ABB RobotStudio station: Demo Solar Simulation.rspag

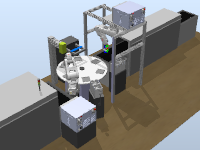
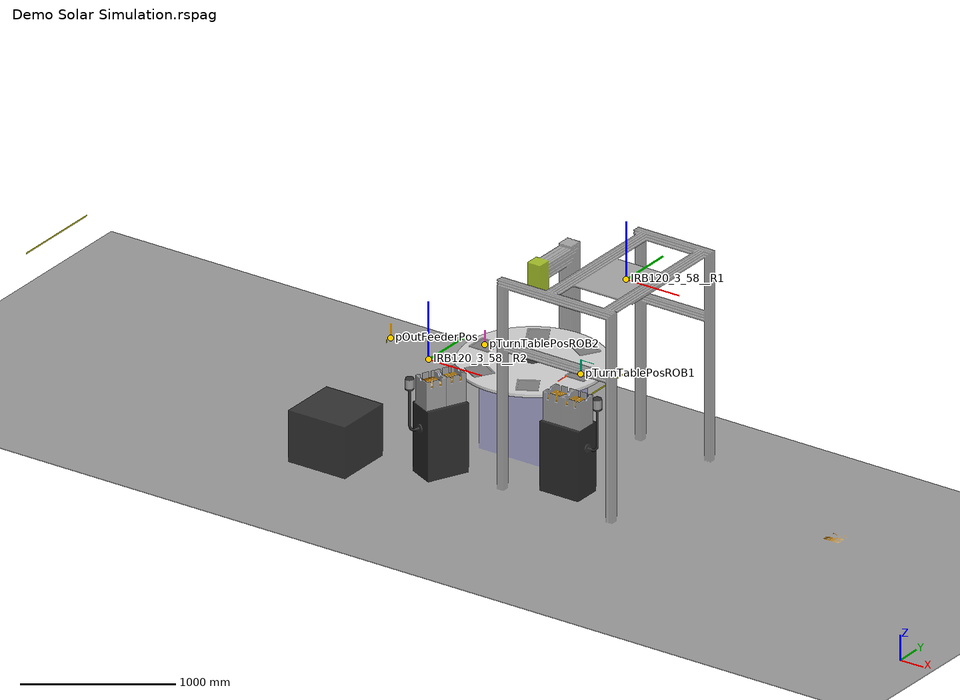
[picture v1: parts stored in the station drawn from their meshes, with robot base, taught points and paths (robot models come from the ABB library and are not in the file)]
--- station ---
Station Demo Solar Simulation (saved by RobotStudio 21.4.9694.0)
Controller IRB120_ROB1, task T_ROB1: task frame (RAPID world) sits at (800, -100, 1439.5) mm, rotated rx 180 ry 0 rz 90 deg in the station
Controller IRB120_ROB2, task T_ROB1: task frame (RAPID world) sits at (-554.4, -372.68, 600) mm, rotated rx 0 ry 0 rz 45 deg in the station
Controller IRB120_ROB2
  mechanical unit ROB_1: IRB120_3_58__R2, 6 joints, base frame (0, 0, 0) mm
Controller IRB120_ROB1
  mechanical unit ROB_1: IRB120_3_58__R1, 6 joints, base frame (0, 0, 0) mm
Layout (positions relative to the parent item):
  - Robotfoot_600 [part, from Libraries\Robotfoot_600.rslib] at (-554.37, -514.08, 0) mm, rotated rx 0 ry 0 rz 45 deg
  - VisionCamStand1 [part] at (-238.48, 626.57, 0) mm, size 100 x 350 x 1120 mm
  - SC_TurnTable [smart component] at (-5618.3, -2219.9, 0) mm
      signals: DI diROB1detached, DI diRotateOK_ROB2, DI diRotateOK_ROB1, DO doTurnTableInPos, DO doCellInPickPosROB2, DO doTurnTableReadyToRotate
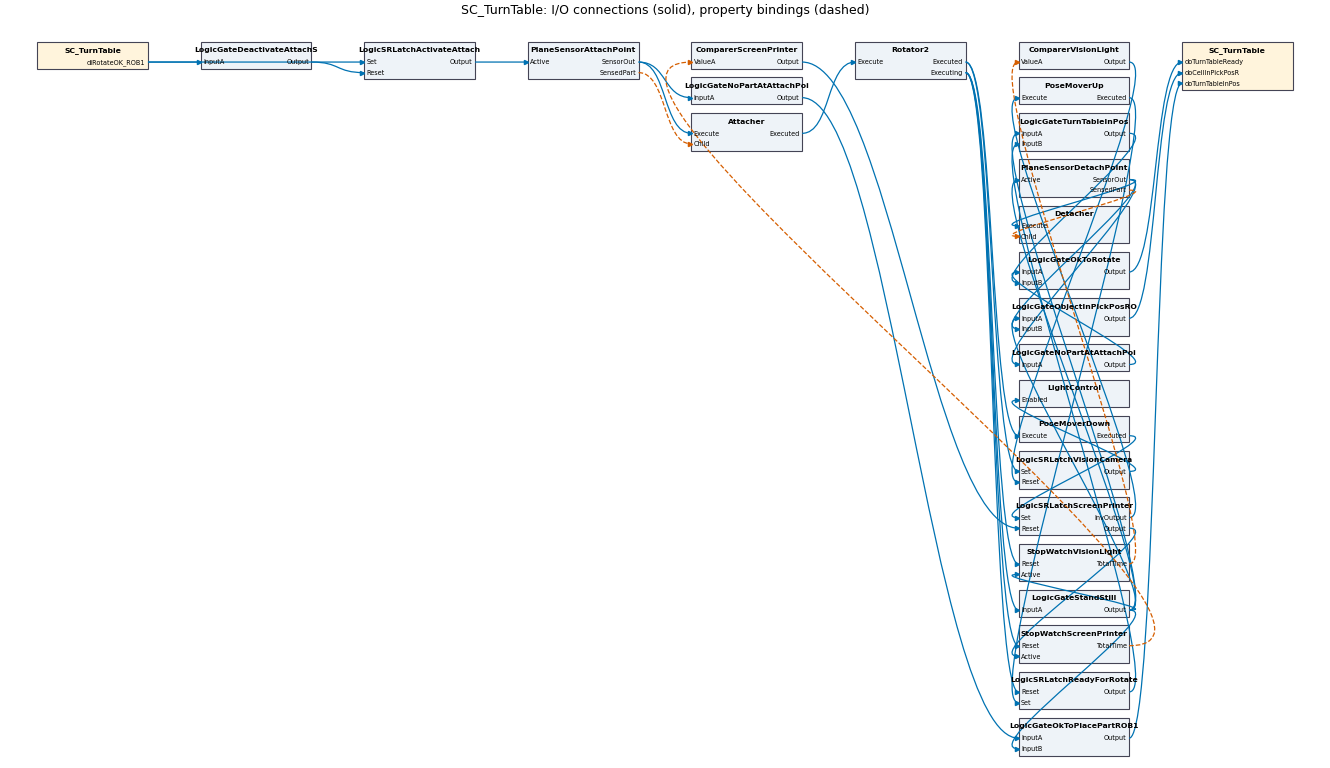
      connections:
        Rotator2.Executed -> PoseMoverDown.Execute
        Rotator2.Executing -> StopWatchVisionLight.Reset
        Rotator2.Executing -> LogicGateStandStill.InputA
        Rotator2.Executed -> LogicSRLatchVisionCamera.Set
        Rotator2.Executing -> StopWatchScreenPrinter.Reset
        Rotator2.Executing -> LogicSRLatchReadyForRotate.Reset
        LogicGateStandStill.Output -> StopWatchVisionLight.Active
        ComparerVisionLight.Output -> LogicSRLatchVisionCamera.Reset
        PoseMoverDown.Executed -> LogicSRLatchScreenPrinter.Set
        ComparerScreenPrinter.Output -> LogicSRLatchScreenPrinter.Reset
        LogicSRLatchScreenPrinter.InvOutput -> PoseMoverUp.Execute
        LogicSRLatchScreenPrinter.Output -> StopWatchScreenPrinter.Active
        PoseMoverUp.Executed -> LogicSRLatchReadyForRotate.Set
        Attacher.Executed -> Rotator2.Execute
        LogicGateStandStill.Output -> LogicGateTurnTableInPos.InputA
        LogicSRLatchReadyForRotate.Output -> LogicGateTurnTableInPos.InputB
        PlaneSensorAttachPoint.SensorOut -> Attacher.Execute
        PlaneSensorDetachPoint.SensorOut -> Detacher.Execute
        LogicGateStandStill.Output -> PlaneSensorDetachPoint.Active
        LogicGateOkToRotate.Output -> SC_TurnTable.doTurnTableReadyToRotate
        LogicSRLatchActivateAttachSensor.Output -> PlaneSensorAttachPoint.Active
        LogicGateStandStill.Output -> LogicGateObjectInPickPosROB2.InputA
        PlaneSensorDetachPoint.SensorOut -> LogicGateObjectInPickPosROB2.InputB
        LogicGateObjectInPickPosROB2.Output -> SC_TurnTable.doCellInPickPosROB2
        PlaneSensorAttachPoint.SensorOut -> LogicGateNoPartAtAttachPoint.InputA
        LogicGateNoPartAtAttachPoint.Output -> LogicGateOkToPlacePartROB1.InputA
        LogicGateStandStill.Output -> LogicGateOkToPlacePartROB1.InputB
        LogicGateOkToPlacePartROB1.Output -> SC_TurnTable.doTurnTableInPos
        PlaneSensorDetachPoint.SensorOut -> LogicGateNoPartAtAttachPointROB2.InputA
        LogicGateNoPartAtAttachPointROB2.Output -> LogicGateOkToRotate.InputA
        LogicGateTurnTableInPos.Output -> LogicGateOkToRotate.InputB
        SC_TurnTable.diRotateOK_ROB1 -> LogicSRLatchActivateAttachSensor.Set
        LogicGateDeactivateAttachSensor.Output -> LogicSRLatchActivateAttachSensor.Reset
        SC_TurnTable.diRotateOK_ROB1 -> LogicGateDeactivateAttachSensor.InputA
        LogicSRLatchVisionCamera.Output -> LightControl.Enabled
        StopWatchVisionLight.TotalTime => ComparerVisionLight.ValueA
        StopWatchScreenPrinter.TotalTime => ComparerScreenPrinter.ValueA
        PlaneSensorAttachPoint.SensedPart => Attacher.Child
        PlaneSensorDetachPoint.SensedPart => Detacher.Child
    - RotatingTable_disc [part] at (5618.3, 2219.9, 580) mm, rotated rx 0 ry 0 rz -120 deg, size 999.8 x 999.8 x 40 mm
    - RotatingTable_base [part] at (5368.3, 1969.9, 0) mm, size 500 x 500 x 580 mm
    - Rotator2 [smart component, from Components\Rotator2.rslib]
        properties: Angle=1.0471975511966; Axis=[0 0 0.001]; CenterPoint=[2.66453525910038E-15 -1.02584607475364E-13 0.579998779296875]; Duration=1; Object=RotatingTable_disc; Reference=Global; ReferenceObject=(none)
    - ScreenPrinter [mechanism] at (5560.76, 2741.46, 0) mm; joint values [0.09] (rad or m)
        links: L1, L2
    - VisionLight2 [part] at (5441.45, 2532.92, 912.77) mm, rotated rx 180 ry 0 rz 180 deg, size 257.1 x 257.1 x 312 mm
    - PoseMoverDown [smart component, from Components\PoseMover.rslib]
        properties: Duration=0.5; Mechanism=ScreenPrinter; Pose=2
    - PoseMoverUp [smart component, from Components\PoseMover.rslib]
        properties: Duration=0.5; Mechanism=ScreenPrinter; Pose=3
    - ComparerVisionLight [smart component, from Components\Comparer.rslib]
        properties: Operator=>=; ValueA=26.0280000000005; ValueB=2
    - StopWatchVisionLight [smart component, from Components\StopWatch.rslib]
        properties: AutoReset=false; LapTime=26.0280000000005; TotalTime=26.0280000000005
    - LogicGateStandStill [smart component, from Components\LogicGate.rslib]
        properties: Delay=0; Operator=NOT
    - Show [smart component, from Components\Show.rslib]
        properties: Object=VisionLight2
    - Hide [smart component, from Components\Hide.rslib]
        properties: Object=VisionLight2
    - ComparerScreenPrinter [smart component, from Components\Comparer.rslib]
        properties: Operator=>=; ValueA=1.008; ValueB=1
    - StopWatchScreenPrinter [smart component, from Components\StopWatch.rslib]
        properties: AutoReset=false; LapTime=1.008; TotalTime=1.008
    - LogicSRLatchScreenPrinter [smart component, from Components\LogicSRLatch.rslib]
    - LogicSRLatchReadyForRotate [smart component, from Components\LogicSRLatch.rslib]
    - Attacher [smart component, from Components\Attacher.rslib]
        properties: Child=(none); Flange=0; Mount=false; Offset=[0 0 0]; Orientation=[0 0 0]; Parent=RotatingTable_disc
    - Detacher [smart component, from Components\Detacher.rslib]
        properties: Child=(none); KeepPosition=true
    - PlaneSensorAttachPoint [smart component, from Components\PlaneSensor.rslib] at (5943.3, 2219.9, 605.5) mm, rotated rx 0 ry -90 rz 0 deg
        properties: Axis1=[0.005 0 0]; Axis2=[0 0.005 0]; Origin=[0 0 0]; SensedPart=(none)
      - _sensorPart_ [part], size 5 x 5 x 0 mm
    - LogicGateTurnTableInPos [smart component, from Components\LogicGate.rslib]
        properties: Delay=0; Operator=AND
    - LogicGateObjectInPickPosROB2 [smart component, from Components\LogicGate.rslib]
        properties: Delay=0; Operator=AND
    - PlaneSensorDetachPoint [smart component, from Components\PlaneSensor.rslib] at (5293.3, 2219.9, 605) mm
        properties: Axis1=[0 0.005 0]; Axis2=[0 0 0.005]; Origin=[0 0 0.0005]; SensedPart=(none)
      - _sensorPart_ [part], size 0 x 5 x 5 mm
    - LogicGateNoPartAtAttachPoint [smart component, from Components\LogicGate.rslib]
        properties: Delay=0; Operator=NOT
    - LogicGateOkToPlacePartROB1 [smart component, from Components\LogicGate.rslib]
        properties: Delay=0; Operator=AND
    - LogicGateNoPartAtAttachPointROB2 [smart component, from Components\LogicGate.rslib]
        properties: Delay=0; Operator=NOT
    - LogicGateOkToRotate [smart component, from Components\LogicGate.rslib]
        properties: Delay=0; Operator=AND
    - LogicSRLatchActivateAttachSensor [smart component, from Components\LogicSRLatch.rslib]
    - LogicGateDeactivateAttachSensor [smart component, from Components\LogicGate.rslib]
        properties: Delay=0; Operator=NOT
    - LogicSRLatchVisionCamera [smart component, from Components\LogicSRLatch.rslib]
    - LightControl [smart component, from Components\LightControl.rslib]
        properties: Light=Spotlight Vision Camera; Color=-65536; CastShadows=true; AmbientIntensity=0; DiffuseIntensity=1; HighlightIntensity=1; SpotAngle=0.366519142918809; Range=0
  - Solar-Ram2 [part] at (790.57, -23.21, 0) mm, size 900 x 1150 x 1500 mm
  - VisionCam [part] at (-138.76, 278.2, 1121.48) mm, rotated rx 180 ry 0 rz 180 deg, size 100 x 100 x 210 mm
  - SC_VacuumGripper_ROB1 [smart component] at (720, 60, 824.5) mm, rotated rx 180 ry 0 rz 0 deg
      properties: DetachedSolarPanel=(none)
      signals: DI diGrip, DO doDetachedROB1, DO doAttached
      connections:
        SC_VacuumGripper_ROB1.diGrip -> PlaneSensor.Active
        PlaneSensor.SensorOut -> Attacher.Execute
        SC_VacuumGripper_ROB1.diGrip -> LogicGateDetach.InputA
        LogicGateDetach.Output -> Detacher.Execute
        Detacher.Executed -> LogicSRLatchDetached.Set
        Attacher.Executed -> LogicSRLatchDetached.Reset
        LogicSRLatchDetached.Output -> SC_VacuumGripper_ROB1.doDetachedROB1
        Attacher.Executed -> LogicSRLatchAttached.Set
        Detacher.Executed -> LogicSRLatchAttached.Reset
        LogicSRLatchAttached.Output -> SC_VacuumGripper_ROB1.doAttached
        PlaneSensor.SensedPart => Attacher.Child
        Attacher.Child => Detacher.Child
        PlaneSensor.SensedPart => SC_VacuumGripper_ROB1.DetachedSolarPanel
    - VacuumGripper [mechanism, from Libraries\VacuumGripper.rslib] at (0, 0, 0) mm
    - PlaneSensor [smart component, from Components\PlaneSensor.rslib]
        properties: Axis1=[0.005 0 0]; Axis2=[0 0 0.002]; Origin=[0 0 0.11501]; SensedPart=(none)
      - _sensorPart_ [part], size 5 x 0 x 2 mm
    - Attacher [smart component, from Components\Attacher.rslib]
        properties: Child=(none); Flange=0; Mount=false; Offset=[0 0 0]; Orientation=[0 0 0]; Parent=VacuumGripper
    - Detacher [smart component, from Components\Detacher.rslib]
        properties: Child=(none); KeepPosition=true
    - LogicGateDetach [smart component, from Components\LogicGate.rslib]
        properties: Delay=0; Operator=NOT
    - LogicSRLatchDetached [smart component, from Components\LogicSRLatch.rslib]
    - LogicSRLatchAttached [smart component, from Components\LogicSRLatch.rslib]
  - SC_VacuumGripper_ROB2 [smart component, from Libraries\SC_VacuumGripper_ROB2.rslib] at (-375, 0, 824) mm, rotated rx 180 ry 0 rz 180 deg
      connections:
        LogicSRLatchAttached.Output -> SC_VacuumGripper_ROB2.doAttached
        Detacher.Executed -> LogicSRLatchAttached.Reset
        Attacher.Executed -> LogicSRLatchAttached.Set
        Attacher.Executed -> LogicSRLatchDetached.Reset
        Detacher.Executed -> LogicSRLatchDetached.Set
        LogicGateDetach.Output -> Detacher.Execute
        SC_VacuumGripper_ROB2.diGrip -> LogicGateDetach.InputA
        PlaneSensorGripperROB2.SensorOut -> Attacher.Execute
        SC_VacuumGripper_ROB2.diGrip -> PlaneSensorGripperROB2.Active
        LogicSRLatchDetached.Output -> SC_VacuumGripper_ROB2.doDetachedROB2
        PlaneSensorGripperROB2.SensedPart => Attacher.Child
        Attacher.Child => Detacher.Child
    - VacuumGripper [mechanism, from Libraries\SC_VacuumGripper_ROB2.rslib] at (0, 0, 0) mm
    - PlaneSensorGripperROB2 [smart component, from Libraries\SC_VacuumGripper_ROB2.rslib]
        properties: Axis1=[0.005 0 0]; Axis2=[0 0 0.002]; Origin=[0 0 0.11501]; SensedPart=(none)
      - _sensorPart_ [part, from Libraries\SC_VacuumGripper_ROB2.rslib]
    - Attacher [smart component, from Libraries\SC_VacuumGripper_ROB2.rslib]
        properties: Child=(none); Flange=0; Mount=false; Offset=[0 0 0]; Orientation=[0 0 0]; Parent=VacuumGripper
    - Detacher [smart component, from Libraries\SC_VacuumGripper_ROB2.rslib]
        properties: Child=(none); KeepPosition=true
    - LogicGateDetach [smart component, from Libraries\SC_VacuumGripper_ROB2.rslib]
        properties: Delay=0; Operator=NOT
    - LogicSRLatchDetached [smart component, from Libraries\SC_VacuumGripper_ROB2.rslib]
    - LogicSRLatchAttached [smart component, from Libraries\SC_VacuumGripper_ROB2.rslib]
  - SC_OutFeeder [smart component, from Libraries\SC_OutFeeder.rslib]
      connections:
        PlaneSensor.SensorOut -> Queue.Delete
        SC_OutFeeder.diPartDetachedROB2 -> Queue.Enqueue
        LineSensor.SensedPart => Queue.Back
    - Solar_FiringFurnace [part, from Libraries\SC_OutFeeder.rslib] at (-2925.68, -654.53, 0) mm
    - LineSensor [smart component, from Components\LineSensor.rslib] at (-925.82, -314.47, 605) mm, rotated rx 0 ry 0 rz -180 deg
        properties: End=[0 0 0.01]; Radius=0.001; SensedPart=(none); SensedPoint=[0 0 0]; Start=[0 0 -0.01]
      - _sensorPart_ [part], size 2 x 2 x 20 mm
    - LinearMover [smart component, from Components\LinearMover.rslib]
        properties: Direction=[-1 0 0]; Object=Queue; Reference=Global; ReferenceObject=(none); Speed=0.5
    - Queue [smart component, from Components\Queue.rslib]
        properties: Back=(none); Front=(none); NumberOfObjects=0; Queue={C5565BCE-F788-4268-B9EA-6DC8EDB4EF1C}
    - PlaneSensor [smart component, from Components\PlaneSensor.rslib] at (-3551.59, -594.57, 607) mm, rotated rx 180 ry 0 rz -180 deg
        properties: Axis1=[0 0 -0.01]; Axis2=[0 0.679 0]; Origin=[0 0 0.006]; SensedPart=(none)
      - _sensorPart_ [part], size 0 x 679 x 10 mm
    - Sink [smart component, from Components\Sink.rslib]
        properties: Object=(none)
  - SC_SolarPanelControlBufferROB1 [smart component]
      signals: DI diDetachedROB1, DO doBufferFull, DO doPlacePanelInBuffer
      connections:
        LineSensor.SensorOut -> QueueBuffer.Enqueue
        LineSensor.SensorOut -> LogicGate.InputA
        SC_SolarPanelControlBufferROB1.diDetachedROB1 -> LogicGate.InputB
        LogicGate.Output -> QueueBuffer.DeleteAll
        LineSensor.SensorOut -> SC_SolarPanelControlBufferROB1.doBufferFull
        Comparer.Output -> SC_SolarPanelControlBufferROB1.doPlacePanelInBuffer
        LineSensor.SensorOut -> Random.Execute
        LineSensor.SensorOut -> StopWatch.Reset
        Comparer.Output -> Highlighter.Active
        Comparer.Output -> LightControl.Enabled
        LineSensor.SensedPart => QueueBuffer.Back
        StopWatch.TotalTime => Comparer.ValueA
        Random.Value => Comparer.ValueB
    - LineSensor [smart component, from Components\LineSensor.rslib] at (535.16, -496.34, 690.45) mm, rotated rx -90 ry 0 rz 0 deg
        properties: End=[0 0 0.01]; Radius=0.001; SensedPart=(none); SensedPoint=[0 0 0]; Start=[0 0 0]
      - _sensorPart_ [part], size 2 x 2 x 10 mm
    - QueueBuffer [smart component, from Components\Queue.rslib]
        properties: Back=(none); Front=(none); NumberOfObjects=2; Queue={5b4a490e-e94d-4e7d-aaa3-7820dbafc272};{f1dc00a8-52dc-4df7-b1a1-4e36716e6d69};{3331a42c-4012-47dd-a22c-2bd2aaf43c34};{22d48996-991e-442b-9ad3-6191d561751a}
    - LogicGate [smart component, from Components\LogicGate.rslib]
        properties: Delay=0; Operator=AND
    - Random [smart component, from Components\Random.rslib]
        properties: Max=30; Min=10; Value=24.2007750525143
    - StopWatch [smart component, from Components\StopWatch.rslib]
        properties: AutoReset=false; LapTime=21.9240000000004; TotalTime=21.9240000000004
    - Comparer [smart component, from Components\Comparer.rslib]
        properties: Operator=>=; ValueA=21.9240000000004; ValueB=24.2007750525143
    - SolarPanelBuffer [part] at (427.16, -333.84, 0) mm, size 300 x 200 x 700 mm
    - MatrixRepeater [smart component, from Components\MatrixRepeater.rslib] at (0, 0, 142) mm
        properties: CountX=2; CountY=1; CountZ=5; OffsetX=0.148; OffsetY=0.1; OffsetZ=0.0041; Source=SolarPanel2
      - SolarPanel2 [part], size 120 x 120 x 4 mm
      - SolarPanel2 [part] at (148, 0, 0) mm, size 120 x 120 x 4 mm
      - SolarPanel2 [part] at (0, 0, 4.1) mm, size 120 x 120 x 4 mm
      - SolarPanel2 [part] at (148, 0, 4.1) mm, size 120 x 120 x 4 mm
      - SolarPanel2 [part] at (0, 0, 8.2) mm, size 120 x 120 x 4 mm
      - SolarPanel2 [part] at (148, 0, 8.2) mm, size 120 x 120 x 4 mm
      - SolarPanel2 [part] at (0, 0, 12.3) mm, size 120 x 120 x 4 mm
      - SolarPanel2 [part] at (148, 0, 12.3) mm, size 120 x 120 x 4 mm
      - SolarPanel2 [part] at (0, 0, 16.4) mm, size 120 x 120 x 4 mm
      - SolarPanel2 [part] at (148, 0, 16.4) mm, size 120 x 120 x 4 mm
    - lamp_buffer1 [part] at (1157.11, 444.56, 0) mm, size 59.9 x 59.9 x 60 mm
    - lamp_stand [part] at (727.16, -433.84, 350) mm, rotated rx 90 ry 0 rz 90 deg, size 60 x 410 x 110 mm
    - Highlighter [smart component, from Components\Highlighter.rslib]
        properties: Color=[255 255 0]; Object=lamp_buffer1; Opacity=240
    - SolarPanel1_1 [part] at (502.66, -433.84, 647.24) mm, rotated rx 0 ry 0 rz 90 deg, size 120 x 120 x 4 mm
    - SolarPanel1_2 [part, from Libraries\SolarPanel1_2.rslib] at (652.66, -433.84, 647.24) mm, rotated rx 0 ry 0 rz 90 deg
    - SolarPanel2 [part], size 120 x 120 x 4 mm
    - LightControl [smart component, from Components\LightControl.rslib]
        properties: Light=Point Light R1; Color=-256; CastShadows=false; AmbientIntensity=0; DiffuseIntensity=0.600000023841858; HighlightIntensity=1; SpotAngle=1.0471975511966; Range=0.3
  - SC_SolarPanelControlBufferROB2 [smart component] at (384.37, -330.21, 0) mm, rotated rx 0 ry 0 rz -115 deg
      signals: DO doBufferFull, DO doPlacePanelInBuffer, DI diDetachedROB2
      connections:
        LineSensorBufferROB2.SensorOut -> StopWatch.Reset
        LineSensorBufferROB2.SensorOut -> Random.Execute
        Comparer.Output -> SC_SolarPanelControlBufferROB2.doPlacePanelInBuffer
        LineSensorBufferROB2.SensorOut -> SC_SolarPanelControlBufferROB2.doBufferFull
        LogicGate.Output -> QueueBuffer.DeleteAll
        SC_SolarPanelControlBufferROB2.diDetachedROB2 -> LogicGate.InputB
        LineSensorBufferROB2.SensorOut -> LogicGate.InputA
        LineSensorBufferROB2.SensorOut -> QueueBuffer.Enqueue
        Comparer.Output -> Highlighter.Active
        Comparer.Output -> LightControl.Enabled
        LineSensorBufferROB2.SensedPart => QueueBuffer.Back
        StopWatch.TotalTime => Comparer.ValueA
        Random.Value => Comparer.ValueB
    - MatrixRepeater [smart component] at (0, 0, 142.05) mm
        properties: CountX=2; CountY=1; CountZ=5; OffsetX=0.148; OffsetY=0; OffsetZ=0.0041; Source=SolarPanel2
      - SolarPanel2 [part], size 120 x 120 x 4 mm
      - SolarPanel2 [part] at (148, 0, 0) mm, size 120 x 120 x 4 mm
      - SolarPanel2 [part] at (0, 0, 4.1) mm, size 120 x 120 x 4 mm
      - SolarPanel2 [part] at (148, 0, 4.1) mm, size 120 x 120 x 4 mm
      - SolarPanel2 [part] at (0, 0, 8.2) mm, size 120 x 120 x 4 mm
      - SolarPanel2 [part] at (148, 0, 8.2) mm, size 120 x 120 x 4 mm
      - SolarPanel2 [part] at (0, 0, 12.3) mm, size 120 x 120 x 4 mm
      - SolarPanel2 [part] at (148, 0, 12.3) mm, size 120 x 120 x 4 mm
    - LineSensorBufferROB2 [smart component] at (535.16, -496.34, 690.45) mm, rotated rx -90 ry 0 rz 0 deg
        properties: End=[0 0 0.01]; Radius=0.001; SensedPart=(none); SensedPoint=[0 0 0]; Start=[0 0 0]
        signals: DI Active, DO SensorOut
      - _sensorPart_ [part], size 2 x 2 x 10 mm
    - QueueBuffer [smart component]
        properties: Back=(none); Front=(none); NumberOfObjects=3; Queue={66f4f5c0-1914-4998-becb-bacfb7656e75};{1fbde2fe-55c7-4f7a-8a39-f6660a833d7e};{27abcaec-d6a0-42b8-b182-1693c2f83687};{973bea39-a09e-4329-ba59-f6a02a91c1a0}
        signals: DI Enqueue, DI Dequeue, DI Clear, DI Delete, DI DeleteAll
    - LogicGate [smart component]
        properties: Delay=0; Operator=AND
        signals: DI InputA, DI InputB, DO Output
    - Random [smart component]
        properties: Max=20; Min=5; Value=17.9851557677543
        signals: DI Execute, DO Executed
    - StopWatch [smart component]
        properties: AutoReset=false; LapTime=23.4960000000004; TotalTime=23.4960000000004
        signals: DI Active, DI Reset, DI Lap
    - Comparer [smart component]
        properties: Operator=>=; ValueA=23.4960000000004; ValueB=17.9851557677543
        signals: DO Output
    - SolarPanelBuffer [part] at (427.16, -333.84, 0) mm, size 300 x 200 x 700 mm
    - lamp_buffer2 [part] at (-136.83, -487.91, 0) mm, rotated rx 0 ry 0 rz 115 deg, size 59.9 x 59.9 x 60 mm
    - lamp_stand [part] at (727.16, -433.84, 350) mm, rotated rx 90 ry 0 rz 90 deg, size 60 x 410 x 110 mm
    - Highlighter [smart component, from Components\Highlighter.rslib]
        properties: Color=[255 255 0]; Object=lamp_buffer2; Opacity=240
    - SolarPanel2_1 [part, from Libraries\SolarPanel2_1.rslib] at (502.66, -433.84, 658.45) mm, rotated rx 0 ry 0 rz 90 deg
    - SolarPanel2_2 [part] at (652.66, -433.84, 658.45) mm, rotated rx 0 ry 0 rz 90 deg, size 120 x 120 x 4 mm
    - LightControl [smart component, from Components\LightControl.rslib]
        properties: Light=Point Light R2; Color=-256; CastShadows=false; AmbientIntensity=0; DiffuseIntensity=0.5; HighlightIntensity=1; SpotAngle=1.0471975511966; Range=0.3
  - ControllerStand [part], size 443 x 426 x 373.8 mm
  - Floor [part], size 8000 x 3000 x 6 mm
  - SC_SolarPanelInFeeder [smart component]
      signals: AO aoOrientation, AO aoPositionY, AO aoPositionX, DO doObjectInPos
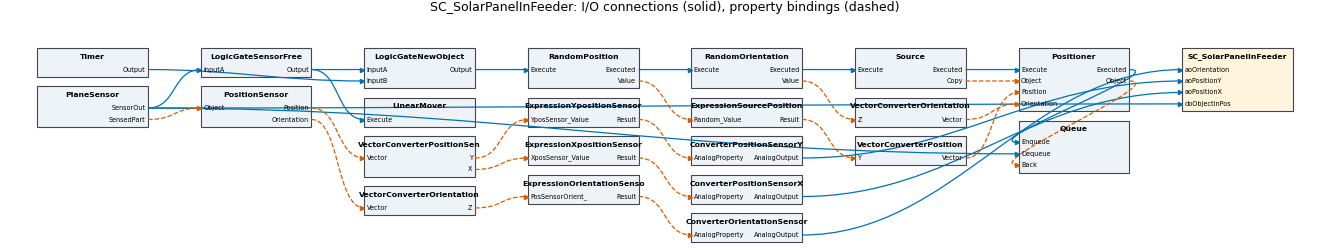
      connections:
        LogicGateSensorFree.Output -> LogicGateNewObject.InputA
        Timer.Output -> LogicGateNewObject.InputB
        LogicGateNewObject.Output -> RandomPosition.Execute
        RandomPosition.Executed -> RandomOrientation.Execute
        RandomOrientation.Executed -> Source.Execute
        Source.Executed -> Positioner.Execute
        PlaneSensor.SensorOut -> LogicGateSensorFree.InputA
        Positioner.Executed -> Queue.Enqueue
        PlaneSensor.SensorOut -> Queue.Dequeue
        LogicGateSensorFree.Output -> LinearMover.Execute
        ConverterOrientationSensor.AnalogOutput -> SC_SolarPanelInFeeder.aoOrientation
        ConverterPositionSensorY.AnalogOutput -> SC_SolarPanelInFeeder.aoPositionY
        ConverterPositionSensorX.AnalogOutput -> SC_SolarPanelInFeeder.aoPositionX
        PlaneSensor.SensorOut -> SC_SolarPanelInFeeder.doObjectInPos
        RandomPosition.Value => ExpressionSourcePosition.Random_Value
        Source.Copy => Positioner.Object
        ExpressionSourcePosition.Result => VectorConverterPosition.Y
        VectorConverterPosition.Vector => Positioner.Position
        RandomOrientation.Value => VectorConverterOrientation.Z
        VectorConverterOrientation.Vector => Positioner.Orientation
        Positioner.Object => Queue.Back
        PlaneSensor.SensedPart => PositionSensor.Object
        PositionSensor.Position => VectorConverterPositionSensor.Vector
        ExpressionYpositionSensor.Result => ConverterPositionSensorY.AnalogProperty
        PositionSensor.Orientation => VectorConverterOrientationSensor.Vector
        VectorConverterOrientationSensor.Z => ExpressionOrientationSensor.PosSensorOrient_Value
        ExpressionOrientationSensor.Result => ConverterOrientationSensor.AnalogProperty
        VectorConverterPositionSensor.Y => ExpressionYpositionSensor.YposSensor_Value
        VectorConverterPositionSensor.X => ExpressionXpositionSensor.XposSensor_Value
        ExpressionXpositionSensor.Result => ConverterPositionSensorX.AnalogProperty
    - Source [smart component, from Components\Source.rslib] at (0, 142.31, 0) mm
        properties: Copy=(none); Orientation=[0 0 0]; Parent=(none); Position=[2.378 0 0.603]; Source=SolarPanel; Transient=true; PhysicsBehavior=0
    - RandomPosition [smart component, from Components\Random.rslib]
        properties: Max=100; Min=-100; Value=-96.6233353114796
    - ExpressionSourcePosition [smart component, from Components\Expression.rslib]
        properties: Expression=(Random_Value)/1000; Random_Value=-96.6233353114796; Result=-0.0966233353114796
    - Positioner [smart component, from Components\Positioner.rslib] at (142.31, 174.78, 0) mm
        properties: Object=(none); Orientation=[0 0 44.0577471391567]; Position=[0 -0.0966233353114796 0]; Reference=Local; ReferenceObject=(none)
    - VectorConverterPosition [smart component, from Components\VectorConverter.rslib]
        properties: Vector=[0 -0.0966233353114796 0]; X=0; Y=-0.0966233353114796; Z=0
    - RandomOrientation [smart component, from Components\Random.rslib]
        properties: Max=45; Min=-45; Value=44.0577471391567
    - VectorConverterOrientation [smart component, from Components\VectorConverter.rslib]
        properties: Vector=[0 0 44.0577471391567]; X=0; Y=0; Z=44.0577471391567
    - PlaneSensor [smart component, from Components\PlaneSensor.rslib]
        properties: Axis1=[0 -0.38 0]; Axis2=[0 0 0.01]; Origin=[0.6 0.18 0.604]; SensedPart=(none)
      - _sensorPart_ [part], size 0 x 380 x 10 mm
    - Timer [smart component, from Components\Timer.rslib]
        properties: CurrentTime=8.112; Interval=3; Repeat=true; StartTime=0
    - LogicGateNewObject [smart component, from Components\LogicGate.rslib]
        properties: Delay=0; Operator=AND
    - LogicGateSensorFree [smart component, from Components\LogicGate.rslib]
        properties: Delay=0; Operator=NOT
    - LinearMover [smart component, from Components\LinearMover.rslib]
        properties: Direction=[-1 0 0]; Object=Queue; Reference=Global; ReferenceObject=(none); Speed=0.25
    - Queue [smart component, from Components\Queue.rslib]
        properties: Back=(none); Front=(none); NumberOfObjects=2; Queue={1853B5AC-4FCE-4C79-973A-8B0D704E15C4};{C0E9B6BD-3140-45EC-A4F6-77C0983F29F9};{96F1CB72-C972-42DC-B470-F6ADD5B15031};{85065212-1676-49A4-B366-2FDB271ED009};{7C824E8E-7F59-4FA9-BE2F-60013457640B};{CBDCE347-6FB3-46D8-B261-28A78DEE33B8};{C95F343E-8BED-44FD-918F-39FFD95E1EF3};{2093C68E-4AFF-431D-A86C-45413FB2F8F8};{05A19856-DC61-4F5F-892B-641957E78D17};{8728EC80-36FA-4B95-84C7-421037A7D638};{80E97431-519E-4202-A655-BA1EA0236438};{4D8C8765-9334-4259-B14A-122944BE8095};{C47A8979-25F7-4A87-91E8-97E12E45B89C};{557234E6-817D-4097-B2F7-91FB90F1C251};{0337C678-C0CB-4C30-9497-F88585278B86};{9A7F6220-568F-4985-AD87-70C2DFC3D232};{4D66CF9A-92F3-45C7-BBF2-C3F850698689};{FCEC3C40-F459-49FD-B11A-8221D654EC0F};{5C56DA9C-0043-4CFF-ACAE-A4EEB87EEC8D};{DCED1F5F-16B4-4AC0-B11D-87AE7AD175A8};{630D608E-57D6-4390-9D61-58657C0654A5};{B4144B91-A2F2-426F-B949-F36246469BE5};{bd42e0d9-1469-474a-812f-c5de7074ceaa};{66f4f5c0-1914-4998-becb-bacfb7656e75};{5b4a490e-e94d-4e7d-aaa3-7820dbafc272};{340e28b5-26bc-4687-b395-17a2afa88c16};{0784914d-9285-4180-b7dc-6d29963e447b};{b25ac926-7d93-4474-96b2-9efd9fe282d1};{f1dc00a8-52dc-4df7-b1a1-4e36716e6d69};{5e703e08-b24e-43c5-9e52-5d17626a8394};{33b902e5-9dcf-4fea-b03b-6281b6d07689};{1fbde2fe-55c7-4f7a-8a39-f6660a833d7e};{27abcaec-d6a0-42b8-b182-1693c2f83687};{9d43facc-f590-4450-bc61-0f1bb3e6d83f};{3331a42c-4012-47dd-a22c-2bd2aaf43c34};{973bea39-a09e-4329-ba59-f6a02a91c1a0};{6c6f2fdb-752d-49b5-809d-3f6e8a1a61ed};{e544f0ad-c5f2-414c-ae96-0da9b34aa504};{22d48996-991e-442b-9ad3-6191d561751a};{beb4460c-9896-43c8-b76c-478cee5d8ca7};{44b7b48d-9f7f-42a9-b69d-8c0b2a5f6734};{f88fddc4-5c71-4644-ab94-2e990e875dc6};{37f61219-1f7b-4fb1-98d6-90da7d8c230a};{dd77935a-2902-4922-990d-0a0a7d2f7b97};{b3d12fd5-70ab-4382-8aca-79ddbca6265c};{cd94ddbb-cd08-4396-87da-7b52593a22e5}
    - PositionSensor [smart component, from Components\PositionSensor.rslib]
        properties: Object=(none); Orientation=[0 0 0.351181464454085]; Position=[0.674000000000025 0.078944081523899 0.603]; Reference=Global; ReferenceObject=(none)
    - VectorConverterPositionSensor [smart component, from Components\VectorConverter.rslib]
        properties: Vector=[0.674000000000025 0.078944081523899 0.603]; X=0.674000000000025; Y=0.078944081523899; Z=0.603
    - ConverterPositionSensorY [smart component, from Components\Converter.rslib]
        properties: AnalogProperty=78.944081523899; BooleanProperty=false; DigitalProperty=0; GroupProperty=0
    - ExpressionYpositionSensor [smart component, from Components\Expression.rslib]
        properties: Expression=YposSensor_Value*1000; Result=78.944081523899; YposSensor_Value=0.078944081523899
    - VectorConverterOrientationSensor [smart component, from Components\VectorConverter.rslib]
        properties: Vector=[0 0 0.351181464454085]; X=0; Y=0; Z=0.351181464454085
    - ConverterOrientationSensor [smart component, from Components\Converter.rslib]
        properties: AnalogProperty=20.1212157564426; BooleanProperty=false; DigitalProperty=0; GroupProperty=0
    - ExpressionOrientationSensor [smart component, from Components\Expression.rslib]
        properties: Expression=PosSensorOrient_Value*(180/pi); PosSensorOrient_Value=0.351181464454085; Result=20.1212157564426
    - ExpressionXpositionSensor [smart component, from Components\Expression.rslib]
        properties: Expression=(XposSensor_Value*1000)-660; Result=14.0000000000249; XposSensor_Value=0.674000000000025
    - ConverterPositionSensorX [smart component, from Components\Converter.rslib]
        properties: AnalogProperty=14.0000000000249; BooleanProperty=false; DigitalProperty=0; GroupProperty=0
    - Solar_Dryer [part, from Libraries\Solar_Dryer.rslib] at (1114.49, -259.61, 0) mm
  - SolarPanel [part] at (2378.83, -8.13, 0) mm, size 120 x 120 x 4 mm
  - IRB120_3_58__R2 [mechanism, from Robots\IRB120_3_58_G_01.rslib] at (-554.4, -372.68, 600) mm, rotated rx 0 ry 0 rz 45 deg; joint values [0.3368, 0.7092, 0.2152, 0, 0.6464, 1.1222] (rad or m)
  - IRB120_3_58__R1 [mechanism, from Robots\IRB120_3_58_G_01.rslib] at (800, -100, 1439.5) mm, rotated rx 180 ry 0 rz 90 deg; joint values [2.6779, -1.7361, 0.679, 0, -0.5137, -1.1071] (rad or m)
  - IRC5_Compact_R2 [part, from Equipment\IRC5_Compact__02.rslib] at (-1136.33, -1115.23, 373.76) mm
  - IRC5_Compact_R1 [part, from Equipment\IRC5_Compact__02.rslib] at (564.47, -673.21, 1500) mm
  - Frame_R1 [frame] at (800, -100, 1439.5) mm, rotated rx 180 ry 0 rz 90 deg
  - Frame_R2 [frame] at (-554.4, -372.68, 600) mm, rotated rx 0 ry 0 rz 45 deg
Attachment: SC_VacuumGripper_ROB1 is attached to IRB120_3_58__R1 / Link6
Attachment: SC_VacuumGripper_ROB2 is attached to IRB120_3_58__R2 / Link6
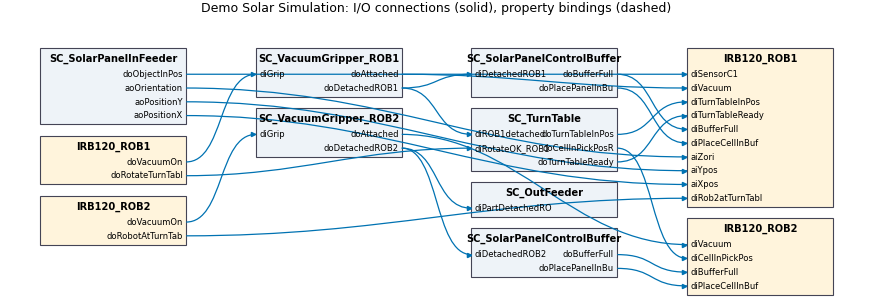
Station logic (signal -> signal, property => property):
  SC_SolarPanelInFeeder.doObjectInPos -> IRB120_ROB1.diSensorC1
  IRB120_ROB1.doVacuumOn -> SC_VacuumGripper_ROB1.diGrip
  SC_VacuumGripper_ROB1.doAttached -> IRB120_ROB1.diVacuum
  SC_VacuumGripper_ROB1.doDetachedROB1 -> SC_TurnTable.diROB1detached
  IRB120_ROB1.doRotateTurnTable -> SC_TurnTable.diRotateOK_ROB1
  SC_TurnTable.doTurnTableInPos -> IRB120_ROB1.diTurnTableInPos
  SC_VacuumGripper_ROB2.doAttached -> IRB120_ROB2.diVacuum
  IRB120_ROB2.doVacuumOn -> SC_VacuumGripper_ROB2.diGrip
  SC_TurnTable.doCellInPickPosROB2 -> IRB120_ROB2.diCellInPickPos
  SC_VacuumGripper_ROB2.doDetachedROB2 -> SC_OutFeeder.diPartDetachedROB2
  SC_TurnTable.doTurnTableReadyToRotate -> IRB120_ROB1.diTurnTableReadyToRotate
  SC_SolarPanelControlBufferROB1.doBufferFull -> IRB120_ROB1.diBufferFull
  SC_SolarPanelControlBufferROB1.doPlacePanelInBuffer -> IRB120_ROB1.diPlaceCellInBuffer
  SC_VacuumGripper_ROB1.doDetachedROB1 -> SC_SolarPanelControlBufferROB1.diDetachedROB1
  SC_SolarPanelControlBufferROB2.doBufferFull -> IRB120_ROB2.diBufferFull
  SC_SolarPanelControlBufferROB2.doPlacePanelInBuffer -> IRB120_ROB2.diPlaceCellInBuffer
  SC_VacuumGripper_ROB2.doDetachedROB2 -> SC_SolarPanelControlBufferROB2.diDetachedROB2
  SC_SolarPanelInFeeder.aoOrientation -> IRB120_ROB1.aiZori
  SC_SolarPanelInFeeder.aoPositionY -> IRB120_ROB1.aiYpos
  SC_SolarPanelInFeeder.aoPositionX -> IRB120_ROB1.aiXpos
  IRB120_ROB2.doRobotAtTurnTable -> IRB120_ROB1.diRob2atTurnTable

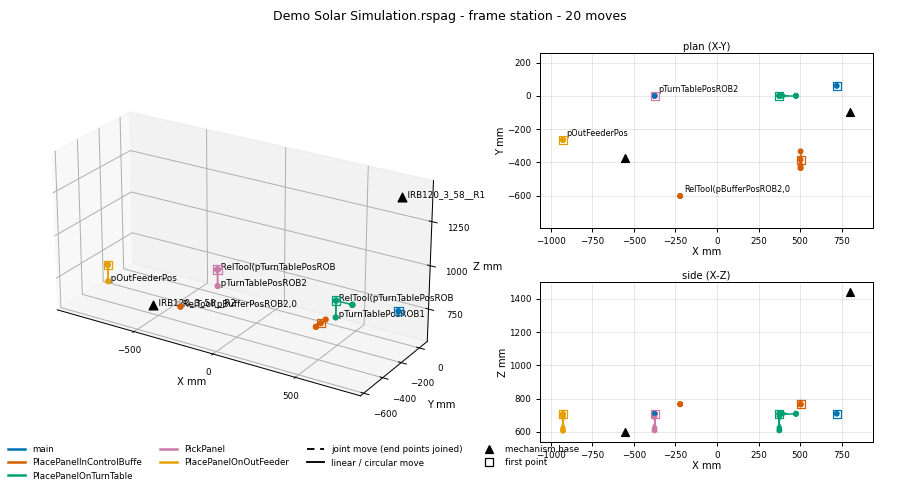
[picture p0: tool path of Demo Solar Simulation.rspag in frame station, 20 of 25 moves have a stored position in this frame; points joined in program order, loops and branches not executed]
--- Backups/IRB120_ROB1/RAPID/TASK1/PROGMOD/modCalibData.mod ---
%%%
   VERSION: 1
   LANGUAGE: ENGLISH
%%%

MODULE modCalibData
	PERS tooldata tGripper:=[TRUE,[[0,0,115],[1,0,0,0]],[1,[0,0,80],[1,0,0,0],0,0,0]];
	PERS wobjdata wobjPickPosC1:=[FALSE,TRUE,"",[[65.4074,-66.6415,834.499],[2.48646E-32,0.991445,-0.130524,-7.7537E-33]],[[0,0,0],[1,0,0,0]]];
	PERS wobjdata wobjPickPosC2:=[FALSE,TRUE,"",[[122.978,-101.908,834.499],[0,0.991445,0.130528,-6.03955E-33]],[[0,0,0],[1,0,0,0]]];
	PERS wobjdata wobjPickPosC3:=[FALSE,TRUE,"",[[-94.661,-117.307,834.499],[2.58483E-32,0.953717,0.300707,3.36101E-32]],[[0,0,0],[1,0,0,0]]];
!	PERS wobjdata wobjPickPos:=[FALSE,TRUE,"",[[75.6855229268255,-140.000000000001,832.49890136719],[-9.65203756683695E-18,1,-1.11022302462516E-16,7.33157456517778E-17]],[[0,0,0],[1,0,0,0]]];
	PERS wobjdata wobjTurnTableROB1:=[FALSE,TRUE,"",[[100,-425,834.5],[2.00306E-16,-0.707107,0.707107,2.00306E-16]],[[0,0,0],[1,0,0,0]]];
	TASK PERS wobjdata wobjBuffer:=[FALSE,TRUE,"",[[-233.842,-72.8418,939.499],[0,-0.707107,0.707107,0]],[[0,0,0],[1,0,0,0]]];
	PERS wobjdata wobjPickPos:=[FALSE,TRUE,"",[[100,-140,832.499],[4.5017E-17,0.707107,0.707107,4.59278E-16]],[[17,-82.0115,0],[0.473135,0,0,-0.88099]]];
	TASK PERS wobjdata wobjPickPosStatic:=[FALSE,TRUE,"",[[100,-140,832.499],[4.5017E-17,0.707107,0.707107,4.59278E-16]],[[0,0,0],[1,0,0,0]]];
ENDMODULE

--- Backups/IRB120_ROB1/RAPID/TASK1/PROGMOD/modRobotStudio.mod ---
MODULE modRobotStudio
	CONST robtarget pPickPosC1:=[[60,60.0000000000002,2.5],[6.12303176911189E-17,1,4.48916032525077E-33,-3.69778549322349E-32],[1,0,-2,5],[9E9,9E9,9E9,9E9,9E9,9E9]];
	CONST robtarget pPickPosC2:=[[60,60.0000000000001,2.5],[-6.12303176911189E-17,1,4.62223186652937E-33,-6.16297582203915E-33],[1,0,-2,5],[9E9,9E9,9E9,9E9,9E9,9E9]];
	CONST robtarget pPickPosC3:=[[60,60.0000000000001,2.5],[-6.12303176911188E-17,1,1.07852076885685E-32,1.23259516440783E-32],[0,0,-1,5],[9E9,9E9,9E9,9E9,9E9,9E9]];
	CONST robtarget pBufferPosROB1:=[[224.500035230802,100.000011574079,166.454416191376],[-8.61528821582825E-16,0.707106781186548,-0.707106781186547,3.72302807738425E-17],[0,0,-1,4],[9E9,9E9,9E9,9E9,9E9,9E9]];
	CONST robtarget pTurnTablePosROB1:=[[0,0,4],[-6.12303176911189E-17,1,-5.55111512312578E-17,-1.97057596545677E-46],[1,0,-3,4],[9E9,9E9,9E9,9E9,9E9,9E9]];
	PERS bool bPartPlacedOnTurnTable:=FALSE;
	PERS num nZoffset:=-16;
	CONST robtarget pPickPos:=[[0,0,0],[-6.12303176911189E-17,1,4.75531733503912E-33,-3.08148791101958E-32],[1,0,-2,5],[9E9,9E9,9E9,9E9,9E9,9E9]];
	PERS bool bWobjCalculated:=FALSE;

PROC main()
	MoveJ RelTool(pPickPosC1,0,0,-100),v200,fine,tGripper\WObj:=wobjPickPosStatic;
	bPartPlacedOnTurnTable:=FALSE;
	nZoffset:=0;
	WHILE TRUE DO
		PickPanel;
		IF diPlaceCellInBuffer=1 THEN
			PlacePanelInControlBuffer;
		ELSE
			PlacePanelOnTurnTable;
		ENDIF
	ENDWHILE
ENDPROC

PROC PickPanel()
	WaitUntil diSensorC1=1 AND bWobjCalculated=TRUE;
	MoveJ RelTool(pPickPos,0,0,-100),v2000,z5,tGripper\WObj:=wobjPickPos;
	MoveL RelTool(pPickPos,0,0,-2),v100,fine,tGripper\WObj:=wobjPickPos;
	SetDO doVacuumOn,1;
	WaitDI diVacuum,1;
	MoveL RelTool(pPickPos,0,0,-100),v500,z50,tGripper\WObj:=wobjPickPos;

ENDPROC

PROC PlacePanelInControlBuffer()
	MoveJ RelTool(pBufferPosROB1,50,0,-100),v1000,z10,tGripper\WObj:=wobjBuffer;
	MoveL RelTool(pBufferPosROB1,0,0,-100),v1000,z1,tGripper\WObj:=wobjBuffer;
	MoveL RelTool(pBufferPosROB1,0,0,nZoffset),v100,fine,tGripper\WObj:=wobjBuffer;
	IF diBufferFull=1 THEN
		nZoffset:=0;
	ELSE
		nZoffset:=nZoffset-4;
	ENDIF
	SetDO doVacuumOn,0;
	WaitDI diVacuum,0;
	MoveL RelTool(pBufferPosROB1,0,0,-100),v100,z1,tGripper\WObj:=wobjBuffer;
	MoveL RelTool(pBufferPosROB1,100,0,-100),v200,fine,tGripper\WObj:=wobjBuffer;
ENDPROC

PROC PlacePanelOnTurnTable()
	MoveJ  RelTool(pTurnTablePosROB1,0,0,-100),v2000,fine,tGripper\WObj:=wobjTurnTableROB1;
	WaitUntil diTurnTableInPos=1 AND bPartPlacedOnTurnTable=FALSE;
	MoveL  pTurnTablePosROB1,v100,fine,tGripper\WObj:=wobjTurnTableROB1;
	SetDO doVacuumOn,0;
	WaitDI diVacuum,0;
	MoveL  RelTool(pTurnTablePosROB1,0,0,-100),v200,z10,tGripper\WObj:=wobjTurnTableROB1;
    IF diSensorC1=1 AND bWobjCalculated=TRUE THEN
	    MoveL  RelTool(pTurnTablePosROB1,-100,0,-100),v1000,z50,tGripper\WObj:=wobjTurnTableROB1;
    ELSE
	    MoveL  RelTool(pTurnTablePosROB1,-100,0,-100),v200,fine,tGripper\WObj:=wobjTurnTableROB1;
    ENDIF
	bPartPlacedOnTurnTable:=TRUE;
ENDPROC
ENDMODULE

--- Backups/IRB120_ROB1/RAPID/TASK1/SYSMOD/LINKEDM.sys ---
%%%
  VERSION:1
  LANGUAGE:ENGLISH
%%%

MODULE LINKEDM (SYSMODULE)

! FOLLOWER
!     Name of electronically linked follower axis used by operator at teach pendent.
      PERS string l_f_axis_name{5}       :=  ["",  "", "", "", ""];

!     Name of the mechanical unit for follower axis.
      PERS string l_f_mecunt_n{5}  :=  ["", "", "", "", ""];

!     Linked follower axis number in the mechanical unit (first axis in mech. unit is number 1).
      PERS num l_f_axis_no{5}      :=  [0,          0,   0,  0,  0];

! MASTER
!     Name of the mechanical unit for linked master axis.
      PERS string l_m_mecunt_n{5} :=  ["", "", "", "", ""];

!     Linked master axis number in the mechanical unit (first axis in mech. unit is number 1).
!     See axis number table in documentation for different master mechanical units.
      PERS num l_m_axis_no{5}     :=  [0,  0,  0,  0,  0];

! POSITION OFFSET
!     The increase of the allowed offset position between the master and follower
!     positions, used when starting AUTO mode. As soon as the offset is decreased
!     the old configurated parameter is used.
!     Example: 3 => the configurated value of allowed offset is increased 3 times.
      PERS num offset_ratio{5}       :=  [10,  10,   10,  10,  10];

! SPEED RATIO
!     Speed_ratio used in AUTO and JOG modes [ very_slow   slow    normal    fast]
!     Value 1 = max allowed manual speed.
      CONST num speed_ratio {20}      := [0.01, 0.01, 0.01, 0.01, 0.01,
                                          0.05, 0.05, 0.05, 0.05, 0.05,
                                          0.20, 0.20, 0.20, 0.20, 0.20,
                                          1.00, 1.00, 1.00, 1.00, 1.00];

! STEP SIZE
!     Displacement position used in JOG mode for each activation of positive or
!     negative movement.                  [very_short    short   normal   long]
!     Unit degees or meter.
      CONST num displacement {20}     := [0.001, 0.001, 0.001, 0.001, 0.001,
                                          0.005, 0.005, 0.005, 0.005, 0.005,
                                          0.020, 0.020, 0.020, 0.020, 0.020,
                                          0.100, 0.100, 0.100, 0.100, 0.100];


!-------------------------------------------------------------
 PROC Linked_m ()
      Linked_m_exe ;
 ENDPROC
ENDMODULE

--- Backups/IRB120_ROB1/RAPID/TASK2/PROGMOD/modTurnTable.mod ---
MODULE modTurnTable
    PERS bool bPartPlacedOnTurnTable:=FALSE;

    PROC main()
        SetDO doRotateTurnTable,0;
        WHILE TRUE DO
            WaitUntil bPartPlacedOnTurnTable=TRUE AND diTurnTableReadyToRotate=1 AND diRob2atTurnTable=0;
            SetDO doRotateTurnTable,1;
            WaitDI diTurnTableInPos,0;
            SetDO doRotateTurnTable,0;
            bPartPlacedOnTurnTable:=FALSE;
        ENDWHILE
    ENDPROC
ENDMODULE

--- Backups/IRB120_ROB1/RAPID/TASK3/PROGMOD/modVisionSimulator.mod ---
MODULE modVisionSimulator
PERS wobjdata wobjPickPos:=[FALSE,TRUE,"",[[100,-140,832.499],[4.5017E-17,0.707107,0.707107,4.59278E-16]],[[17,-82.0115,0],[0.473135,0,0,-0.88099]]];
TASK PERS wobjdata wobjPickPosStatic:=[FALSE,TRUE,"",[[100,-140.000000000001,832.49890136719],[4.50170397023425E-17,0.707106781186548,0.707106781186547,4.59278319577846E-16]],[[0,0,0],[1,0,0,0]]];
PERS bool bWobjCalculated:=FALSE;

PROC main()
bWobjCalculated:=FALSE;
WHILE TRUE DO
	WaitDI diSensorC1,1;
	CalculateWobj;
	WaitDI diSensorC1,0;
	bWobjCalculated:=FALSE;
ENDWHILE
ENDPROC

PROC CalculateWobj()
wobjPickPos:=wobjPickPosStatic;
wobjPickPos.oframe.trans.x:=aiXpos;
wobjPickPos.oframe.trans.y:=aiYpos;
wobjPickPos.oframe.rot:=OrientZYX(aiZori,0,0);
bWobjCalculated:=TRUE;
ENDPROC
ENDMODULE

--- Backups/IRB120_ROB2/RAPID/TASK1/PROGMOD/modCalibData.mod ---
%%%
   VERSION: 1
   LANGUAGE: ENGLISH
%%%

MODULE modCalibData
	PERS tooldata tGripper:=[TRUE,[[0,0,115],[1,0,0,0]],[1,[0,0,80],[1,0,0,0],0,0,0]];
	TASK PERS wobjdata wobjTurnTableROB2:=[FALSE,TRUE,"",[[390.377,136.672,4.99878],[0.382684,-5.00251E-32,5.6752E-31,0.92388]],[[0,0,0],[1,0,0,0]]];
	TASK PERS wobjdata wobjOutFeeder:=[FALSE,TRUE,"",[[238.11,480.52,6.10352E-05],[0.38268,0,0,0.923881]],[[0,0,0],[1,0,0,0]]];
	TASK PERS wobjdata wobjBuffer:=[FALSE,TRUE,"",[[-103.652,-568.77,-100],[0.984808,0,0,0.173648]],[[0,0,0],[1,0,0,0]]];
ENDMODULE

--- Backups/IRB120_ROB2/RAPID/TASK1/PROGMOD/modRobotStudio.mod ---
MODULE modRobotStudio
    CONST robtarget pTurnTablePosROB2:=[[0,4.89842541528954E-16,4],[-6.12303176911189E-17,1,-1.61279309130843E-47,0],[0,0,0,0],[9E9,9E9,9E9,9E9,9E9,9E9]];
    CONST robtarget pOutFeederPos:=[[200.016009205003,399.937244742038,6.99993896484363],[-2.01362528565985E-22,0.999999999994593,3.28860826072754E-06,-6.12303176907878E-17],[1,0,1,0],[9E9,9E9,9E9,9E9,9E9,9E9]];
    CONST robtarget pBufferPosROB2:=[[224.500035230801,100.00001157408,166.454416191376],[4.32963728535968E-17,0.707106781186547,0.707106781186548,4.32963728535968E-17],[-1,0,-1,0],[9E9,9E9,9E9,9E9,9E9,9E9]];
    PERS num nZoffset:=-20;



    PROC PickPanel()
        IF diCellInPickPos=0 THEN
            MoveJ RelTool(pTurnTablePosROB2,0,0,-100),v1000,fine,tGripper\WObj:=wobjTurnTableROB2;
            WaitDI diCellInPickPos,1;
        ELSE
            MoveJ RelTool(pTurnTablePosROB2,0,0,-100),v1000,z100,tGripper\WObj:=wobjTurnTableROB2;
        ENDIF
        SetDO doRobotAtTurnTable,1;
        MoveL pTurnTablePosROB2,v200,fine,tGripper\WObj:=wobjTurnTableROB2;
        SetDO doVacuumOn,1;
        WaitDI diVacuum,1;
        MoveLDO RelTool(pTurnTablePosROB2,0,0,-100),v200,z10,tGripper\WObj:=wobjTurnTableROB2,doRobotAtTurnTable,0;
    ENDPROC

    PROC PlacePanelInControlBuffer()
        MoveJ RelTool(pBufferPosROB2,0,0,-100),v1000,z10,tGripper\WObj:=wobjBuffer;
        MoveL RelTool(pBufferPosROB2,0,0,nZoffset),v100,fine,tGripper\WObj:=wobjBuffer;
        IF diBufferFull=1 THEN
            nZoffset:=0;
        ELSE
            nZoffset:=nZoffset-4;
        ENDIF
        SetDO doVacuumOn,0;
        WaitDI diVacuum,0;
        MoveL RelTool(pBufferPosROB2,0,0,-100),v1000,z10,tGripper\WObj:=wobjBuffer;
    ENDPROC

    PROC PlacePanelOnOutFeeder()
        MoveJ RelTool(pOutFeederPos,0,0,-100),v1000,z10,tGripper\WObj:=wobjOutFeeder;
        MoveL pOutFeederPos,v200,fine,tGripper\WObj:=wobjOutFeeder;
        SetDO doVacuumOn,0;
        WaitDI diVacuum,0;
        MoveL RelTool(pOutFeederPos,0,0,-100),v1000,z10,tGripper\WObj:=wobjOutFeeder;
    ENDPROC

    PROC main()
        MoveJ RelTool(pTurnTablePosROB2,0,0,-100),v200,fine,tGripper\WObj:=wobjTurnTableROB2;
        nZoffset:=0;
        WHILE TRUE DO
            PickPanel;
            IF diPlaceCellInBuffer=1 THEN
                PlacePanelInControlBuffer;
            ELSE
                PlacePanelOnOutFeeder;
            ENDIF
        ENDWHILE
    ENDPROC
ENDMODULE

--- Backups/IRB120_ROB1/SYSPAR/EIO.cfg ---
EIO:CFG_1.0:6:1::
#
EIO_SIGNAL:

      -Name "diSensorC1" -SignalType "DI" -Access "All"

      -Name "diSensorC2" -SignalType "DI" -Access "All"

      -Name "diSensorC3" -SignalType "DI" -Access "All"

      -Name "diVacuum" -SignalType "DI" -Access "All"

      -Name "diTurnTableInPos" -SignalType "DI" -Access "All"

      -Name "doVacuumOn" -SignalType "DO" -Access "All"

      -Name "doRotateTurnTable" -SignalType "DO" -Access "All"

      -Name "diRob2atTurnTable" -SignalType "DI" -Access "All"

      -Name "diCellAtPickPosROB2" -SignalType "DI" -Access "All"

      -Name "diTurnTableReadyToRotate" -SignalType "DI" -Access "All"

      -Name "diPlaceCellInBuffer" -SignalType "DI" -Access "All"

      -Name "diBufferFull" -SignalType "DI" -Access "All"

      -Name "aiXpos" -SignalType "AI" -Access "All" -MaxLog 1000 -MaxPhys 1000\
      -MaxPhysLimit 1000 -MaxBitVal 1000 -MinLog -1000 -MinPhys -1000\
      -MinPhysLimit -1000 -MinBitVal -1000 -Size 32

      -Name "aiYpos" -SignalType "AI" -Access "All" -MaxLog 1000 -MaxPhys 1000\
      -MaxPhysLimit 1000 -MaxBitVal 1000 -MinLog -1000 -MinPhys -1000\
      -MinPhysLimit -1000 -MinBitVal -1000 -Size 32

      -Name "aiZori" -SignalType "AI" -Access "All" -MaxLog 1000 -MaxPhys 1000\
      -MaxPhysLimit 1000 -MaxBitVal 1000 -MinLog -1000 -MinPhys -1000\
      -MinPhysLimit -1000 -MinBitVal -1000 -Size 32

--- Backups/IRB120_ROB2/SYSPAR/EIO.cfg ---
EIO:CFG_1.0:6:1::
#
EIO_SIGNAL:

      -Name "diVacuum" -SignalType "DI" -Access "All"

      -Name "diCellInPickPos" -SignalType "DI" -Access "All"

      -Name "doVacuumOn" -SignalType "DO" -Access "All"

      -Name "doRobotAtTurnTable" -SignalType "DO" -Access "All"

      -Name "diPlaceCellInBuffer" -SignalType "DI" -Access "All"

      -Name "diBufferFull" -SignalType "DI" -Access "All"
